% RSLogix 500 project JBT BIN_villa_park_fillmore_bin_scrubber_may_13_2020.RSS, saved by version 11.00.00.00 %
PROJECT "JBT BIN"    % processor: MicroLogix 1200 %

PROGRAM FILES
  LAD 2   50 rungs

DATA FILES
  O0 OUTPUT  4 elements
  I1 INPUT  4 elements
  S2 STATUS  66 elements
  B3 BINARY  3 elements
  T4 TIMER  10 elements
  C5 COUNTER  1 elements
  R6 CONTROL  1 elements
  N7 INTEGER  3 elements
  F8 FLOAT  1 elements

LADDER 2
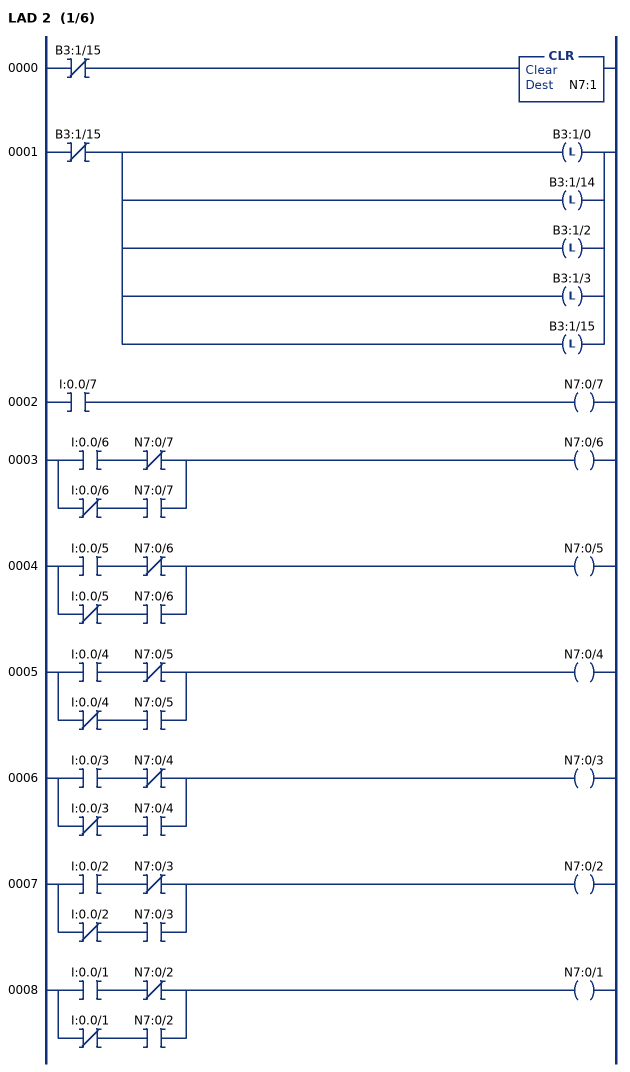
% Rung: 0 %
SOR XIO B3:1/15 CLR N7:1 EOR
% Rung: 1 %
SOR XIO B3:1/15 BST BST OTL B3:1/0 NXB BST OTL B3:1/14 NXB BST OTL B3:1/2 NXB OTL B3:1/3 BND BND BND NXB OTL B3:1/15 BND EOR
% Rung: 2 %
SOR XIC I:0.0/7 OTE N7:0/7 EOR
% Rung: 3 %
SOR BST XIC I:0.0/6 XIO N7:0/7 NXB XIO I:0.0/6 XIC N7:0/7 BND OTE N7:0/6 EOR
% Rung: 4 %
SOR BST XIC I:0.0/5 XIO N7:0/6 NXB XIO I:0.0/5 XIC N7:0/6 BND OTE N7:0/5 EOR
% Rung: 5 %
SOR BST XIC I:0.0/4 XIO N7:0/5 NXB XIO I:0.0/4 XIC N7:0/5 BND OTE N7:0/4 EOR
% Rung: 6 %
SOR BST XIC I:0.0/3 XIO N7:0/4 NXB XIO I:0.0/3 XIC N7:0/4 BND OTE N7:0/3 EOR
% Rung: 7 %
SOR BST XIC I:0.0/2 XIO N7:0/3 NXB XIO I:0.0/2 XIC N7:0/3 BND OTE N7:0/2 EOR
% Rung: 8 %
SOR BST XIC I:0.0/1 XIO N7:0/2 NXB XIO I:0.0/1 XIC N7:0/2 BND OTE N7:0/1 EOR

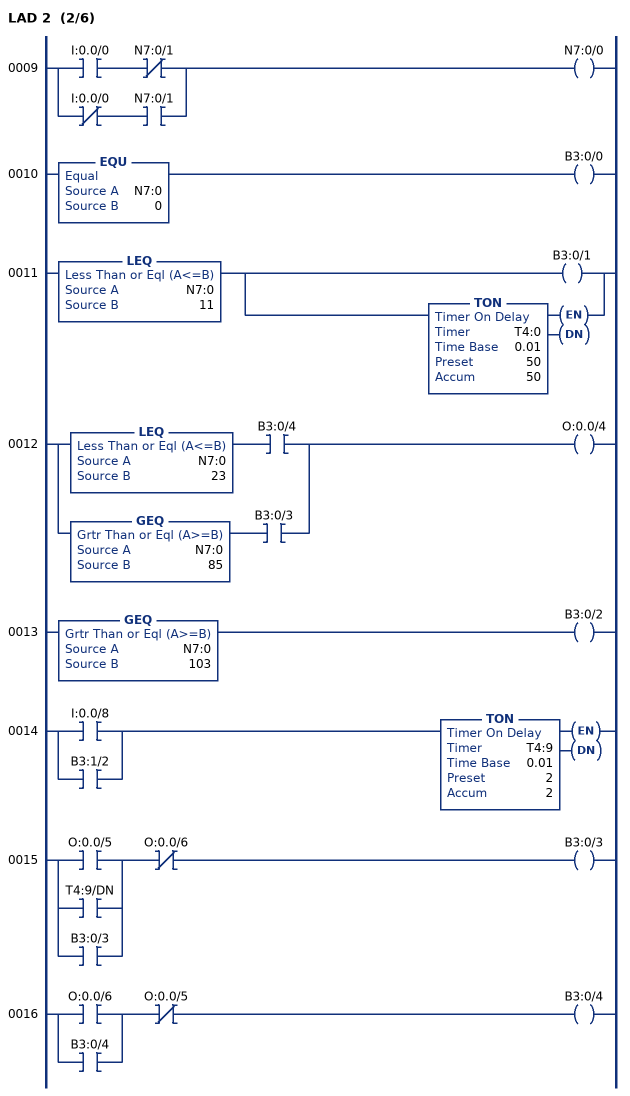
% Rung: 9 %
SOR BST XIC I:0.0/0 XIO N7:0/1 NXB XIO I:0.0/0 XIC N7:0/1 BND OTE N7:0/0 EOR
% Rung: 10 %
SOR EQU N7:0 0 OTE B3:0/0 EOR
% Rung: 11 %
SOR LEQ N7:0 11 BST OTE B3:0/1 NXB TON T4:0 0.01 50 50 BND EOR
% Rung: 12 %
SOR BST LEQ N7:0 23 XIC B3:0/4 NXB GEQ N7:0 85 XIC B3:0/3 BND OTE O:0.0/4 EOR
% Rung: 13 %
SOR GEQ N7:0 103 OTE B3:0/2 EOR
% Rung: 14 %
SOR BST XIC I:0.0/8 NXB XIC B3:1/2 BND TON T4:9 0.01 2 2 EOR
% Rung: 15 %
SOR BST XIC O:0.0/5 NXB XIC T4:9/DN NXB XIC B3:0/3 BND XIO O:0.0/6 OTE B3:0/3 EOR
% Rung: 16 %
SOR BST XIC O:0.0/6 NXB XIC B3:0/4 BND XIO O:0.0/5 OTE B3:0/4 EOR

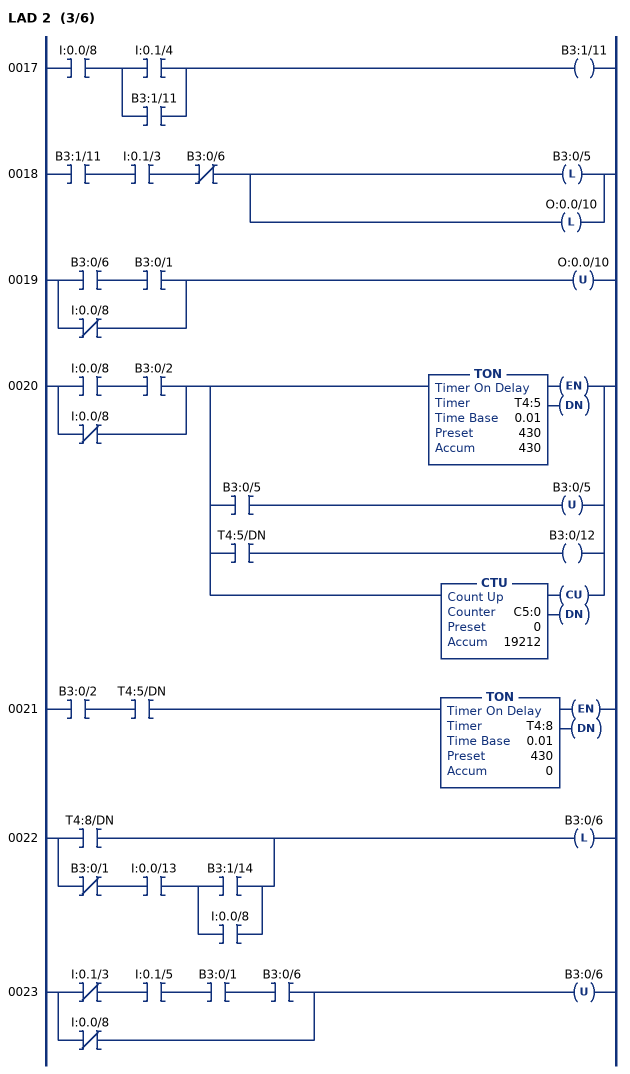
% Rung: 17 %
SOR XIC I:0.0/8 BST XIC I:0.1/4 NXB XIC B3:1/11 BND OTE B3:1/11 EOR
% Rung: 18 %
SOR XIC B3:1/11 XIC I:0.1/3 XIO B3:0/6 BST OTL B3:0/5 NXB OTL O:0.0/10 BND EOR
% Rung: 19 %
SOR BST XIC B3:0/6 XIC B3:0/1 NXB XIO I:0.0/8 BND OTU O:0.0/10 EOR
% Rung: 20 %
SOR BST XIC I:0.0/8 XIC B3:0/2 NXB XIO I:0.0/8 BND BST TON T4:5 0.01 430 430 NXB XIC B3:0/5 OTU B3:0/5 NXB BST XIC T4:5/DN OTE B3:0/12 NXB CTU C5:0 0 19212 BND BND EOR
% Rung: 21 %
SOR XIC B3:0/2 XIC T4:5/DN TON T4:8 0.01 430 0 EOR
% Rung: 22 %
SOR BST XIC T4:8/DN NXB XIO B3:0/1 XIC I:0.0/13 BST XIC B3:1/14 NXB XIC I:0.0/8 BND BND OTL B3:0/6 EOR
% Rung: 23 %
SOR BST XIO I:0.1/3 XIC I:0.1/5 XIC B3:0/1 XIC B3:0/6 NXB XIO I:0.0/8 BND OTU B3:0/6 EOR

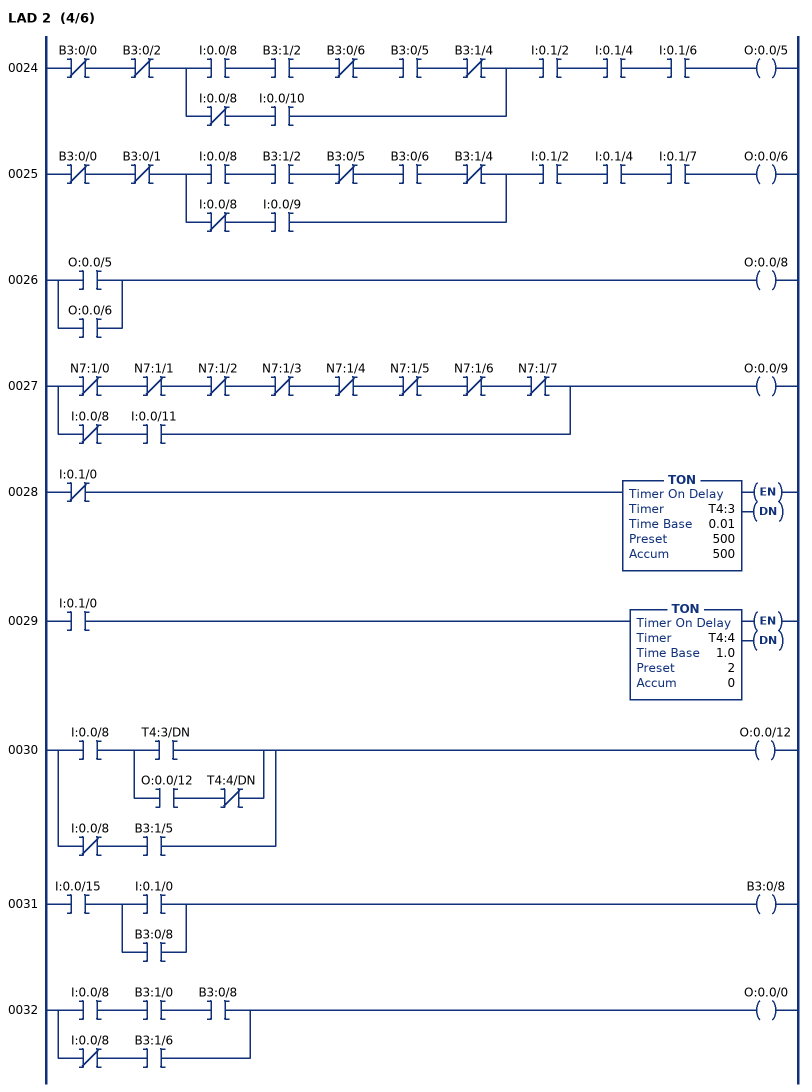
% Rung: 24 %
SOR XIO B3:0/0 XIO B3:0/2 BST XIC I:0.0/8 XIC B3:1/2 XIO B3:0/6 XIC B3:0/5 XIO B3:1/4 NXB XIO I:0.0/8 XIC I:0.0/10 BND XIC I:0.1/2 XIC I:0.1/4 XIC I:0.1/6 OTE O:0.0/5 EOR
% Rung: 25 %
SOR XIO B3:0/0 XIO B3:0/1 BST XIC I:0.0/8 XIC B3:1/2 XIO B3:0/5 XIC B3:0/6 XIO B3:1/4 NXB XIO I:0.0/8 XIC I:0.0/9 BND XIC I:0.1/2 XIC I:0.1/4 XIC I:0.1/7 OTE O:0.0/6 EOR
% Rung: 26 %
SOR BST XIC O:0.0/5 NXB XIC O:0.0/6 BND OTE O:0.0/8 EOR
% Rung: 27 %
SOR BST XIO N7:1/0 XIO N7:1/1 XIO N7:1/2 XIO N7:1/3 XIO N7:1/4 XIO N7:1/5 XIO N7:1/6 XIO N7:1/7 NXB XIO I:0.0/8 XIC I:0.0/11 BND OTE O:0.0/9 EOR
% Rung: 28 %
SOR XIO I:0.1/0 TON T4:3 0.01 500 500 EOR
% Rung: 29 %
SOR XIC I:0.1/0 TON T4:4 1.0 2 0 EOR
% Rung: 30 %
SOR BST XIC I:0.0/8 BST XIC T4:3/DN NXB XIC O:0.0/12 XIO T4:4/DN BND NXB XIO I:0.0/8 XIC B3:1/5 BND OTE O:0.0/12 EOR
% Rung: 31 %
SOR XIC I:0.0/15 BST XIC I:0.1/0 NXB XIC B3:0/8 BND OTE B3:0/8 EOR
% Rung: 32 %
SOR BST XIC I:0.0/8 XIC B3:1/0 XIC B3:0/8 NXB XIO I:0.0/8 XIC B3:1/6 BND OTE O:0.0/0 EOR

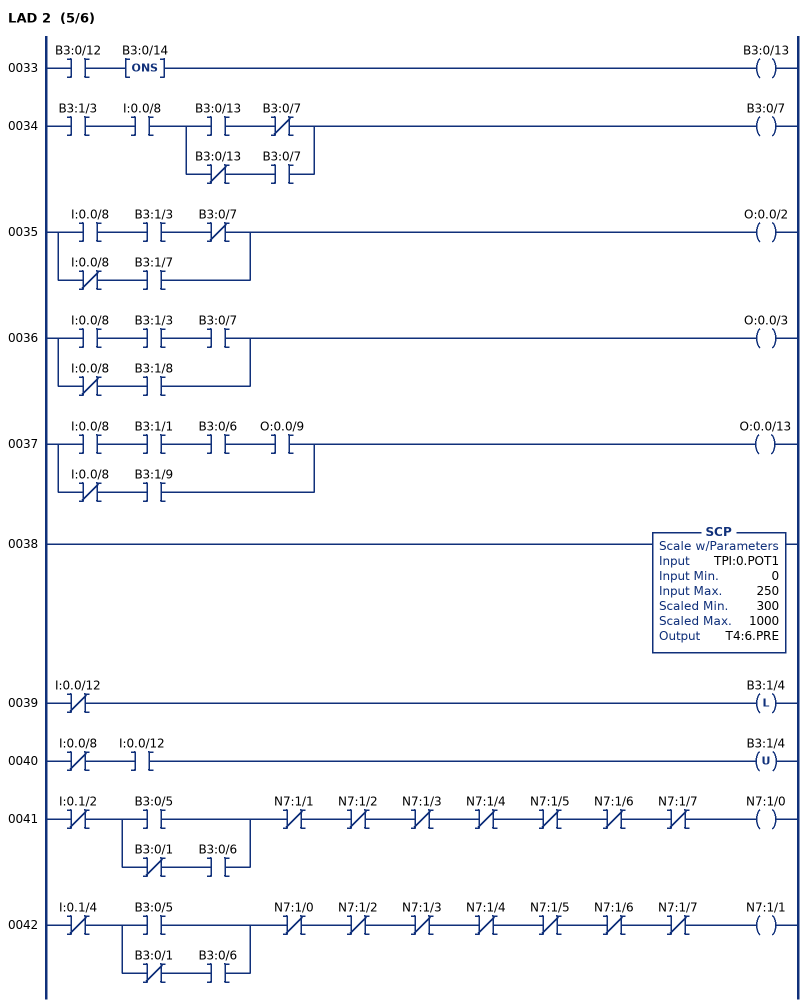
% Rung: 33 %
SOR XIC B3:0/12 ONS B3:0/14 OTE B3:0/13 EOR
% Rung: 34 %
SOR XIC B3:1/3 XIC I:0.0/8 BST XIC B3:0/13 XIO B3:0/7 NXB XIO B3:0/13 XIC B3:0/7 BND OTE B3:0/7 EOR
% Rung: 35 %
SOR BST XIC I:0.0/8 XIC B3:1/3 XIO B3:0/7 NXB XIO I:0.0/8 XIC B3:1/7 BND OTE O:0.0/2 EOR
% Rung: 36 %
SOR BST XIC I:0.0/8 XIC B3:1/3 XIC B3:0/7 NXB XIO I:0.0/8 XIC B3:1/8 BND OTE O:0.0/3 EOR
% Rung: 37 %
SOR BST XIC I:0.0/8 XIC B3:1/1 XIC B3:0/6 XIC O:0.0/9 NXB XIO I:0.0/8 XIC B3:1/9 BND OTE O:0.0/13 EOR
% Rung: 38 %
SOR SCP TPI:0.POT1 0 250 300 1000 T4:6.PRE EOR
% Rung: 39 %
SOR XIO I:0.0/12 OTL B3:1/4 EOR
% Rung: 40 %
SOR XIO I:0.0/8 XIC I:0.0/12 OTU B3:1/4 EOR
% Rung: 41 %
SOR XIO I:0.1/2 BST XIC B3:0/5 NXB XIO B3:0/1 XIC B3:0/6 BND XIO N7:1/1 XIO N7:1/2 XIO N7:1/3 XIO N7:1/4 XIO N7:1/5 XIO N7:1/6 XIO N7:1/7 OTE N7:1/0 EOR
% Rung: 42 %
SOR XIO I:0.1/4 BST XIC B3:0/5 NXB XIO B3:0/1 XIC B3:0/6 BND XIO N7:1/0 XIO N7:1/2 XIO N7:1/3 XIO N7:1/4 XIO N7:1/5 XIO N7:1/6 XIO N7:1/7 OTE N7:1/1 EOR

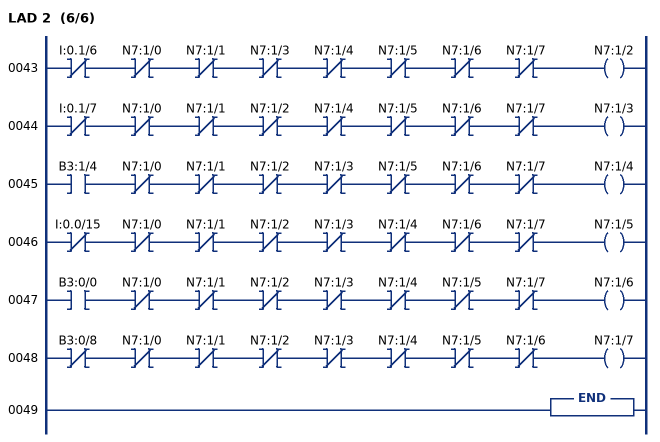
% Rung: 43 %
SOR XIO I:0.1/6 XIO N7:1/0 XIO N7:1/1 XIO N7:1/3 XIO N7:1/4 XIO N7:1/5 XIO N7:1/6 XIO N7:1/7 OTE N7:1/2 EOR
% Rung: 44 %
SOR XIO I:0.1/7 XIO N7:1/0 XIO N7:1/1 XIO N7:1/2 XIO N7:1/4 XIO N7:1/5 XIO N7:1/6 XIO N7:1/7 OTE N7:1/3 EOR
% Rung: 45 %
SOR XIC B3:1/4 XIO N7:1/0 XIO N7:1/1 XIO N7:1/2 XIO N7:1/3 XIO N7:1/5 XIO N7:1/6 XIO N7:1/7 OTE N7:1/4 EOR
% Rung: 46 %
SOR XIO I:0.0/15 XIO N7:1/0 XIO N7:1/1 XIO N7:1/2 XIO N7:1/3 XIO N7:1/4 XIO N7:1/6 XIO N7:1/7 OTE N7:1/5 EOR
% Rung: 47 %
SOR XIC B3:0/0 XIO N7:1/0 XIO N7:1/1 XIO N7:1/2 XIO N7:1/3 XIO N7:1/4 XIO N7:1/5 XIO N7:1/7 OTE N7:1/6 EOR
% Rung: 48 %
SOR XIO B3:0/8 XIO N7:1/0 XIO N7:1/1 XIO N7:1/2 XIO N7:1/3 XIO N7:1/4 XIO N7:1/5 XIO N7:1/6 OTE N7:1/7 EOR
% Rung: 49 %
SOR END EOR

DATA TABLE (non-zero values as saved)
DATA B3
% B3:0 % 0X5D1A 0XC20F 0X8000
DATA T4
% .PRE .ACC %
% T4:0 % 50 50
% T4:1 % 1 0
% T4:2 % 1 0
% T4:3 % 500 500
% T4:4 % 2 0
% T4:5 % 430 430
% T4:6 % 670 0
% T4:7 % 375 500
% T4:8 % 430 0
% T4:9 % 2 2
DATA C5
% .PRE .ACC %
% C5:0 % 0 19212
DATA N7
% N7:0 % 10 0 0
